// TIA Portal V16 export
// export: Created 2023-08-28T09:37:49.80075Z, ExportSetting WithDefaults, DisplayName Totally Integrated Automation Portal, DisplayVersion V16 Update 6, DisplayName TIA Portal Version Control Interface, DisplayVersion V16 Update 2, DisplayName TIA Portal Openness, DisplayVersion V16 Update 6, DisplayName STEP 7 Professional, DisplayVersion V16 Update 6, DisplayName STEP 7 Safety, DisplayVersion V16, DisplayName WinCC Advanced, DisplayVersion V16 Update 6
DATA_BLOCK "operating_mode_select_aut-man_DB"   // DB119
AUTHOR : rtecmer
VERSION : 0.1
// stored: AutoNumber true, DBAccessibleFromOPCUA true, InstanceOfName 08_C_operating_mode_select_aut-man, InstanceOfType FB
"08_C_operating_mode_select_aut-man"
   // VAR
   //    setTrig_M1 : Bool;
   //    setTrig_M2 : Bool;
   //    setTrig_M3 : Bool;
   //    setTrig_M4 : Bool;
   //    setTrig_Z11 : Bool;
   //    setTrig_Z12 : Bool;
   //    set_aut_man_M1 : Bool;
   //    set_aut_man_M2 : Bool;
   //    set_aut_man_M3 : Bool;
   //    set_aut_man_M4 : Bool;
   //    set_aut_man_Z11 : Bool;
   //    set_aut_man_Z12 : Bool;
   // END_VAR
BEGIN
END_DATA_BLOCK
